FUNCTION TryConvert_DATE_TO_ULINT : BOOL
VAR_INPUT
	in : DATE;
	out : REFERENCE TO ULINT;
END_VAR

out := DATE_TO_ULINT(in);
TryConvert_DATE_TO_ULINT := TRUE;

END_FUNCTION

(* stored: Version 1.1.0.1, ProductVersion 3.1.4024.12
   POU TryConvert_DATE_TO_ULINT: Id {015200cb-b751-4d57-a0b6-26967dbcf103}, SpecialFunc None *)
